(* IEC 61131-3 sources: volt/packages/volt-lsp-iec/test-corpus/pro2193/Device/Plc Logic/Application/09 Misc/Library Manager/CAA CiA405, 33 files *)

(* ---- CANOPEN_KERNEL_ERROR.dut ---- *)
TYPE CANOPEN_KERNEL_ERROR :
(
	CANOPEN_KERNEL_NO_ERROR := ANYNUM_TO_WORD(CS.CANOPEN_KERNEL_ERROR.CANOPEN_KERNEL_NO_ERROR),
	CANOPEN_KERNEL_OTHER_ERROR := ANYNUM_TO_WORD(CS.CANOPEN_KERNEL_ERROR.CANOPEN_KERNEL_OTHER_ERROR),
	CANOPEN_KERNEL_DATA_OVERFLOW := ANYNUM_TO_WORD(CS.CANOPEN_KERNEL_ERROR.CANOPEN_KERNEL_DATA_OVERFLOW),
	CANOPEN_KERNEL_TIMEOUT := ANYNUM_TO_WORD(CS.CANOPEN_KERNEL_ERROR.CANOPEN_KERNEL_TIMEOUT),
	CANOPEN_KERNEL_CANBUS_OFF := ANYNUM_TO_WORD(CS.CANOPEN_KERNEL_ERROR.CANOPEN_KERNEL_CANBUS_OFF),
	CANOPEN_KERNEL_CAN_ERROR_PASSIVE := ANYNUM_TO_WORD(CS.CANOPEN_KERNEL_ERROR.CANOPEN_KERNEL_CAN_ERROR_PASSIVE),
	CANOPEN_INTERNAL_FB_ERROR := ANYNUM_TO_WORD(CS.CANOPEN_KERNEL_ERROR.CANOPEN_INTERNAL_FB_ERROR),
	CANOPEN_NO_MORE_MEMORY := ANYNUM_TO_WORD(CS.CANOPEN_KERNEL_ERROR.CANOPEN_NO_MORE_MEMORY),
	CANOPEN_WRONG_PARAMETER := ANYNUM_TO_WORD(CS.CANOPEN_KERNEL_ERROR.CANOPEN_WRONG_PARAMETER),
	CANOPEN_NODEID_UNKNOWN := ANYNUM_TO_WORD(CS.CANOPEN_KERNEL_ERROR.CANOPEN_NODEID_UNKNOWN),
	CANOPEN_NETID_UNKNOWN := ANYNUM_TO_WORD(CS.CANOPEN_KERNEL_ERROR.CANOPEN_NETID_UNKNOWN),
	CANOPEN_REQUEST_ERROR := ANYNUM_TO_WORD(CS.CANOPEN_KERNEL_ERROR.CANOPEN_REQUEST_ERROR),
	CANOPEN_SDOCHANNEL_UNKNOWN := ANYNUM_TO_WORD(CS.CANOPEN_KERNEL_ERROR.CANOPEN_SDOCHANNEL_UNKNOWN),
	CANOPEN_NO_DRIVER := ANYNUM_TO_WORD(CS.CANOPEN_KERNEL_ERROR.CANOPEN_NO_DRIVER),
	CANOPEN_CONFIGURATION_ERROR := ANYNUM_TO_WORD(CS.CANOPEN_KERNEL_ERROR.CANOPEN_CONFIGURATION_ERROR),
	CANOPEN_GUARDING_ERROR := ANYNUM_TO_WORD(CS.CANOPEN_KERNEL_ERROR.CANOPEN_GUARDING_ERROR)
);
END_TYPE

(* ---- DEVICE.dut ---- *)
TYPE DEVICE : USINT (0..127);
END_TYPE

(* ---- DEVICE_STATE.dut ---- *)
TYPE DEVICE_STATE :
(
	INIT,
	RESET_COMM,
	RESET_APP,
	PRE_OPERATIONAL,
	STOPPED,
	OPERATIONAL,
	UNKNOWN,
	NOT_AVAIL
);
END_TYPE

(* ---- EMCY_ERROR.dut ---- *)
TYPE EMCY_ERROR :
STRUCT
	DWDUMMY : DWORD;
	EMCY_ERROR_CODE : WORD;
	ERROR_REGISTER : BYTE;
	BYDUMMY : BYTE;
	ERROR_FIELD : ARRAY [1..5] OF BYTE;
END_STRUCT
END_TYPE

(* ---- SDO_ERROR.dut ---- *)
TYPE SDO_ERROR : UDINT;
END_TYPE

(* ---- SDO_MODE.dut ---- *)
TYPE SDO_MODE :
(
	AUTO := ANYNUM_TO_INT(CS.SDO_MODE.AUTO),
	EXPEDITED := ANYNUM_TO_INT(CS.SDO_MODE.EXPEDITED),
	SEGMENTED := ANYNUM_TO_INT(CS.SDO_MODE.SEGMENTED),
	BLOCK := ANYNUM_TO_INT(CS.SDO_MODE.BLOCK)
);
END_TYPE

(* ---- TRANSITION_STATE.dut ---- *)
TYPE TRANSITION_STATE :
(
	START_REMOTE_NODE := 16#5,
	STOP_REMOTE_NODE := 16#4,
	ENTER_PRE_OPERATIONAL := 16#7F,
	RESET_NODE := 16#6,
	RESET_COMMUNICATION := 16#7,
	ALL_EXCEPT_NMT_AND_SENDER := 16#800
);
END_TYPE

(* ---- CANOPEN_KERNEL_ERROR_CODES.gvl ---- *)
VAR_GLOBAL
	CANOPEN_KERNEL_NO_ERROR : WORD := 16#0;
	CANOPEN_KERNEL_OTHER_ERROR : WORD := 16#1;
	CANOPEN_KERNEL_DATA_OVERFLOW : WORD := 16#2;
	CANOPEN_KERNEL_TIMEOUT : WORD := 16#3;
	CANOPEN_KERNEL_CANBUS_OFF : WORD := 16#10;
	CANOPEN_KERNEL_CAN_ERROR_PASSIVE : WORD := 16#11;
	CANOPEN_INTERNAL_FB_ERROR : WORD := 16#21;
END_VAR

(* ---- GLOBALVARIABLES.gvl ---- *)
VAR_GLOBAL
	GC_USIMAXNETID : USINT := CO.gc_usiMaxNetId;
	GC_USIMAXFBCYCLES : USINT := 4;
	GC_USITIMEOUTPERCENTAGE : USINT := 10;
END_VAR

(* ---- SVN_INFO_FLAGS.gvl ---- *)
VAR_GLOBAL
	XINCOMPLETE : BOOL := FALSE;
	XMODIFIED : BOOL := TRUE;
	XSWITCHED : BOOL := FALSE;
	XCLEAN : BOOL := FALSE;
	XDISCONNECTED : BOOL := FALSE;
END_VAR

(* ---- SVN_INFO_LASTCHANGE.gvl ---- *)
VAR_GLOBAL
	DTLASTCHANGEUTC : DATE_AND_TIME := DATE_AND_TIME#2021-2-4-15:22:35;
	WSLASTCHANGELOCAL : WSTRING(44) := "2021-02-04 16:22:35 +0100 (Thu, 04 Feb 2021)";
	WSLASTCHANGEAUTHOR : WSTRING(8) := "b.schurr";
END_VAR

(* ---- SVN_INFO_REVISIONS.gvl ---- *)
VAR_GLOBAL
	LIMINREVISION : LINT := LINT#52494;
	LIMAXREVISION : LINT := LINT#52494;
END_VAR

(* ---- SVN_INFO_SUMMARY.gvl ---- *)
VAR_GLOBAL
	SVERSIONSUMMARY : STRING(6) := '52494M';
END_VAR

(* ---- SVN_INFO_SUMMARYW.gvl ---- *)
VAR_GLOBAL
	WSVERSIONSUMMARY : WSTRING(6) := "52494M";
END_VAR

(* ---- SVN_INFO_URI.gvl ---- *)
VAR_GLOBAL
	WURL : WSTRING(92) := "svn://server04/LibrariesV3Source/branches/V3.5.17.0/Application/CAA/CAA CiA 405/CAA CiA 405/";
END_VAR

(* ---- GETLIBVERSION.pou ---- *)
FUNCTION GETLIBVERSION : VERSION
END_FUNCTION

(* ---- GETLIBVERSIONNUMBER.pou ---- *)
FUNCTION GETLIBVERSIONNUMBER : DWORD
END_FUNCTION

(* ---- GETSUPPLIERVERSION.pou ---- *)
FUNCTION GETSUPPLIERVERSION : WORD
END_FUNCTION

(* ---- ISLIBRELEASED.pou ---- *)
FUNCTION ISLIBRELEASED : BOOL
END_FUNCTION

(* ---- MAPERROR.pou ---- *)
FUNCTION MAPERROR : CANOPEN_KERNEL_ERROR
VAR_INPUT
	IERROR : INT;
END_VAR
END_FUNCTION

(* ---- CIA405BASE.pou ---- *)
FUNCTION_BLOCK CIA405BASE
VAR_INPUT
	NETWORK : USINT := 1;
	ENABLE : BOOL := FALSE;
	TIMEOUT : UDINT := 0;
END_VAR
VAR_OUTPUT
	CONFIRM : BOOL := FALSE;
	ERROR : CANOPEN_KERNEL_ERROR := CANOPEN_KERNEL_ERROR.CANOPEN_KERNEL_NO_ERROR;
END_VAR
VAR
	XPREVIOUSENABLE : BOOL := FALSE;
	XABORTINPROGRESS : BOOL := FALSE;
	XBUSY : BOOL := FALSE;
	TKSTART : CAA.TICK;
	TKTIMEOUT : CAA.TICK;
	TKACTTIME : CAA.TICK;
	EPROCSTATE : CS.PROC_STATE;
	EPROCCMD : CS.PROC_CMD;
	EERROR : CS.ERROR;
END_VAR
END_FUNCTION_BLOCK

METHOD PRVCYCLICACTION
END_METHOD

METHOD PRVABORT
END_METHOD

METHOD PRVRESETFB
END_METHOD

METHOD PRVSETOUTPUT
VAR_INPUT
	EERR : CANOPEN_KERNEL_ERROR;
END_VAR
END_METHOD

METHOD PRVSTART
END_METHOD

(* ---- GET_CANOPEN_KERNEL_STATE.pou ---- *)
FUNCTION_BLOCK GET_CANOPEN_KERNEL_STATE EXTENDS CiA405Base
VAR_OUTPUT
	STATE : CANOPEN_KERNEL_ERROR := CANOPEN_KERNEL_ERROR.CANOPEN_KERNEL_NO_ERROR;
END_VAR
VAR
	SDO : CS.SDO_READ;
END_VAR
END_FUNCTION_BLOCK

METHOD PRVRESETFB
END_METHOD

METHOD PRVSETOUTPUT
VAR_INPUT
	EERR : CANOPEN_KERNEL_ERROR;
END_VAR
END_METHOD

METHOD PRVSTART
END_METHOD

METHOD PRVCYCLICACTION
END_METHOD

(* ---- GET_LOCAL_NODE_ID.pou ---- *)
FUNCTION_BLOCK GET_LOCAL_NODE_ID EXTENDS CiA405Base
VAR_OUTPUT
	DEVICE : DEVICE := 0;
END_VAR
VAR
	STKINFO : CS.STK_INFO;
END_VAR
END_FUNCTION_BLOCK

METHOD PRVRESETFB
END_METHOD

METHOD PRVSETOUTPUT
VAR_INPUT
	EERR : CANOPEN_KERNEL_ERROR;
END_VAR
END_METHOD

METHOD PRVSTART
END_METHOD

METHOD PRVCYCLICACTION
END_METHOD

(* ---- GET_STATE.pou ---- *)
FUNCTION_BLOCK GET_STATE EXTENDS CiA405Base
VAR_INPUT
	DEVICE : DEVICE := 0;
END_VAR
VAR_OUTPUT
	STATE : DEVICE_STATE := 0;
END_VAR
VAR
	SDO : CS.SDO_READ;
	USIDATA : USINT;
END_VAR
END_FUNCTION_BLOCK

METHOD PRVCYCLICACTION
END_METHOD

METHOD PRVRESETFB
END_METHOD

METHOD PRVSETOUTPUT
VAR_INPUT
	EERR : CANOPEN_KERNEL_ERROR;
END_VAR
END_METHOD

METHOD PRVSTART
END_METHOD

(* ---- NMT.pou ---- *)
FUNCTION_BLOCK NMT EXTENDS CiA405Base
VAR_INPUT
	DEVICE : DEVICE := 0;
	STATE : TRANSITION_STATE := 0;
END_VAR
VAR
	SDO : CS.SDO_WRITE;
	STATEGETTER : GET_STATE;
	BYDATA : BYTE := 0;
END_VAR
END_FUNCTION_BLOCK

METHOD PRVCYCLICACTION
END_METHOD

METHOD PRVRESETFB
END_METHOD

METHOD PRVSTART
END_METHOD

(* ---- RECV_EMCY.pou ---- *)
FUNCTION_BLOCK RECV_EMCY EXTENDS CiA405Base
VAR_OUTPUT
	DEVICE : DEVICE := 0;
	ERRORINFO : EMCY_ERROR;
END_VAR
VAR
	SDO : CS.SDO_READ;
	DATA : CS.EMCY_DATA;
END_VAR
END_FUNCTION_BLOCK

METHOD PRVSTART
END_METHOD

METHOD PRVCYCLICACTION
END_METHOD

METHOD PRVRESETFB
END_METHOD

METHOD PRVSETOUTPUT
VAR_INPUT
	EERR : CANOPEN_KERNEL_ERROR;
END_VAR
END_METHOD

(* ---- RECV_EMCY_DEV.pou ---- *)
FUNCTION_BLOCK RECV_EMCY_DEV EXTENDS CiA405Base
VAR_INPUT
	DEVICE : DEVICE := 0;
END_VAR
VAR_OUTPUT
	ERRORINFO : EMCY_ERROR;
END_VAR
VAR
	SDO : CS.SDO_READ;
	DATA : CS.EMCY_ERROR;
END_VAR
END_FUNCTION_BLOCK

METHOD PRVRESETFB
END_METHOD

METHOD PRVSETOUTPUT
VAR_INPUT
	EERR : CANOPEN_KERNEL_ERROR;
END_VAR
END_METHOD

METHOD PRVSTART
END_METHOD

METHOD PRVCYCLICACTION
END_METHOD

(* ---- SDO_READ.pou ---- *)
FUNCTION_BLOCK SDO_READ EXTENDS CiA405Base
VAR_INPUT
	DEVICE : DEVICE;
	CHANNEL : USINT := 1;
	INDEX : WORD;
	SUBINDEX : BYTE;
	DATA : POINTER TO BYTE;
END_VAR
VAR_OUTPUT
	ERRORINFO : SDO_ERROR;
END_VAR
VAR_IN_OUT
	DATALENGTH : UINT;
END_VAR
VAR
	READ : SDO_READ_DATA;
	UDIDATALENGTH : UDINT;
END_VAR
END_FUNCTION_BLOCK

(* ---- SDO_READ4.pou ---- *)
FUNCTION_BLOCK SDO_READ4 EXTENDS CiA405Base
VAR_INPUT
	DEVICE : DEVICE;
	CHANNEL : USINT := 1;
	INDEX : WORD;
	SUBINDEX : BYTE;
END_VAR
VAR_OUTPUT
	DATA : ARRAY [1..4] OF BYTE;
	DATALENGTH : USINT;
	ERRORINFO : SDO_ERROR;
END_VAR
VAR
	ABYDUMMY : ARRAY [0..2] OF BYTE;
	SDO : CS.SDO_READ;
	PERMISSIONREQUESTSDO : CS.SDO_READ;
	EPERMISSIONREQUEST : CS.PROC_STATE;
	USISDOPERMITTED : USINT;
END_VAR
END_FUNCTION_BLOCK

METHOD PRVABORT
END_METHOD

METHOD PRVRESETFB
END_METHOD

METHOD PRVSETOUTPUT
VAR_INPUT
	EERR : CANOPEN_KERNEL_ERROR;
END_VAR
END_METHOD

METHOD PRVSTART
END_METHOD

METHOD PRVCYCLICACTION
END_METHOD

(* ---- SDO_READ_DATA.pou ---- *)
FUNCTION_BLOCK SDO_READ_DATA EXTENDS CiA405Base
VAR_INPUT
	DEVICE : DEVICE;
	CHANNEL : USINT := 1;
	INDEX : WORD;
	SUBINDEX : BYTE;
	MODE : SDO_MODE := SDO_MODE.AUTO;
	DATA : POINTER TO BYTE;
END_VAR
VAR_OUTPUT
	ERRORINFO : SDO_ERROR;
END_VAR
VAR_IN_OUT
	DATALENGTH : UDINT;
END_VAR
VAR
	SDO : CS.SDO_READ;
	PERMISSIONREQUESTSDO : CS.SDO_READ;
	USISDOPERMITTED : USINT;
	EPERMISSIONREQUEST : CS.PROC_STATE;
END_VAR
END_FUNCTION_BLOCK

METHOD PRVCYCLICACTION
END_METHOD

METHOD PRVABORT
END_METHOD

METHOD PRVRESETFB
END_METHOD

METHOD PRVSETOUTPUT
VAR_INPUT
	EERR : CANOPEN_KERNEL_ERROR;
END_VAR
END_METHOD

METHOD PRVSTART
END_METHOD

(* ---- SDO_WRITE.pou ---- *)
FUNCTION_BLOCK SDO_WRITE EXTENDS CiA405Base
VAR_INPUT
	DEVICE : DEVICE;
	CHANNEL : USINT := 1;
	INDEX : WORD;
	SUBINDEX : BYTE;
	MODE : SDO_MODE;
	DATA : POINTER TO BYTE;
	DATALENGTH : UINT;
END_VAR
VAR_OUTPUT
	ERRORINFO : SDO_ERROR;
END_VAR
VAR
	WRITE : SDO_WRITE_DATA;
END_VAR
END_FUNCTION_BLOCK

(* ---- SDO_WRITE4.pou ---- *)
FUNCTION_BLOCK SDO_WRITE4 EXTENDS CiA405Base
VAR_INPUT
	DEVICE : DEVICE;
	CHANNEL : USINT := 1;
	INDEX : WORD;
	SUBINDEX : BYTE;
	DATA : ARRAY [1..4] OF BYTE;
	DATALENGTH : USINT;
END_VAR
VAR_OUTPUT
	ERRORINFO : SDO_ERROR;
END_VAR
VAR
	ABYDUMMY : ARRAY [0..2] OF BYTE;
	SDO : CS.SDO_WRITE;
	PERMISSIONREQUESTSDO : CS.SDO_READ;
	USISDOPERMITTED : USINT;
	EPERMISSIONREQUEST : CS.PROC_STATE;
END_VAR
END_FUNCTION_BLOCK

METHOD PRVRESETFB
END_METHOD

METHOD PRVSETOUTPUT
VAR_INPUT
	EERR : CANOPEN_KERNEL_ERROR;
END_VAR
END_METHOD

METHOD PRVSTART
END_METHOD

METHOD PRVCYCLICACTION
END_METHOD

METHOD PRVABORT
END_METHOD

(* ---- SDO_WRITE_DATA.pou ---- *)
FUNCTION_BLOCK SDO_WRITE_DATA EXTENDS CiA405Base
VAR_INPUT
	DEVICE : DEVICE;
	CHANNEL : USINT := 1;
	INDEX : WORD;
	SUBINDEX : BYTE;
	MODE : SDO_MODE := SDO_MODE.AUTO;
	DATA : POINTER TO BYTE;
	DATALENGTH : UDINT;
END_VAR
VAR_OUTPUT
	ERRORINFO : SDO_ERROR;
END_VAR
VAR
	SDO : CS.SDO_WRITE;
	PERMISSIONREQUESTSDO : CS.SDO_READ;
	EPERMISSIONREQUEST : CS.PROC_STATE;
	USISDOPERMITTED : USINT;
END_VAR
END_FUNCTION_BLOCK

METHOD PRVCYCLICACTION
END_METHOD

METHOD PRVABORT
END_METHOD

METHOD PRVRESETFB
END_METHOD

METHOD PRVSETOUTPUT
VAR_INPUT
	EERR : CANOPEN_KERNEL_ERROR;
END_VAR
END_METHOD

METHOD PRVSTART
END_METHOD
